INTERFACE I_MessageData

PROPERTY DirRoot : POINTER to string(255)
SET
END_SET
END_PROPERTY

PROPERTY ErrorIndex : reference to uint
SET
END_SET
END_PROPERTY

PROPERTY FileRoot : pointer to string(255)
SET
END_SET
END_PROPERTY

PROPERTY LocalTime : pointer to DT
SET
END_SET
END_PROPERTY

PROPERTY MessageIndex : reference to uint
SET
END_SET
END_PROPERTY

PROPERTY MsgList : pointer to ARRAY[1..GVL_MSG.MAX_MESSAGE] OF st_message
SET
END_SET
END_PROPERTY

END_INTERFACE

(* stored: Version 1.1.0.1, ProductVersion 3.1.4026.18
   Itf I_MessageData: Id {5176a3e7-2d60-4af9-b415-21f1a2a8e77a}
   Property DirRoot: Id {b2af3dbc-8775-41ff-b11d-6c1fa9d1fae9}
   Set Set: Id {125ffdb3-ca6d-4602-be75-c4ab527a807a}
   Property ErrorIndex: Id {2e56a0e8-9e11-4be4-ab04-b877fe4979a9}
   Set Set: Id {28552193-75e6-4eb0-a920-e67ef57c3716}
   Property FileRoot: Id {5cf68986-7e63-4a99-828f-29d0d816b94c}
   Set Set: Id {76593c02-9659-4a5d-bc1a-a560909838c6}
   Property LocalTime: Id {65d5001e-2ba1-47c1-90b0-634b6d0e99c3}
   Set Set: Id {7f1b5ed3-50d5-44cc-9830-a281f17e068e}
   Property MessageIndex: Id {f55ce7c0-2318-46b0-8663-7c2d3b61423f}
   Set Set: Id {a84f3e2f-6958-4ec6-8a91-5a6de4ff6a1f}
   Property MsgList: Id {30bcb3f1-9473-4143-8dcc-eb1ce3a22dfc}
   Set Set: Id {5fc6e1a6-ea93-4fba-9260-05f846a570bf} *)
